FUNCTION_BLOCK PUMP_MDL (* Simple Pump Animation Model *)
  (* Standard: 61499-1 *)
  (* Version 0.2, 2001-04-24, JHC, Rockwell Automation, Moved to fb.rt.process. *)
  (* Version 0.1, 2000-06-21, JHC, Rockwell Automation, Uses LibraryElement.dtd *)
  (* Version 0.0, 2000-05-01, JHC, Rockwell Automation *)
  (* Compiler header: package fb.rt.process; *)
  (* Compiler Java IBM VisualAge 3.0 *)
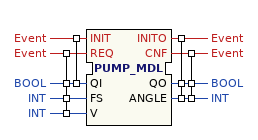
  EVENT_INPUT
    INIT WITH QI; (* Initialization Request *)
    REQ WITH QI, FS, V; (* Simulation Increment *)
  END_EVENT
  EVENT_OUTPUT
    INITO WITH QO, ANGLE; (* Initialization Confirm *)
    CNF WITH QO, ANGLE; (* Increment Confirmation *)
  END_EVENT
  VAR_INPUT
    QI : BOOL; (* Input event qualifier *)
    FS : INT; (* Full-scale speed,degrees per increment *)
    V : INT; (* Angular velocity,percent of FS *)
  END_VAR
  VAR_OUTPUT
    QO : BOOL; (* Output event qualifier *)
    ANGLE : INT; (* Pump Shaft Angle *)
  END_VAR
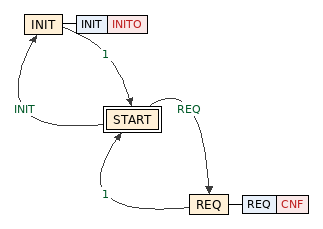
  EC_STATES
    START; (* Initial State *)
    INIT : INIT -> INITO; (* Initialization *)
    REQ : REQ -> CNF; (* Normal execution *)
  END_STATES
  EC_TRANSITIONS
    START TO INIT := INIT;
    INIT TO START := 1;
    START TO REQ := REQ;
    REQ TO START := 1;
  END_TRANSITIONS
  ALGORITHM INIT IN ST:
QO:=QI;

 ANGLE:=0;
  END_ALGORITHM
  ALGORITHM REQ IN ST:
QO:=QI;

 IF QI THEN

 ANGLE:=(ANGLE+FS*V/100)MOD 360;

 END_IF
  END_ALGORITHM
END_FUNCTION_BLOCK
